// TIA Portal project "Project1" (V15.1)

(* hardware
DEVICE "S71500/ET200MP station_1"  S7-1500 station
   slot 0: "PS 25W 24VDC_1"  PS 25W 24VDC  6ES7 505-0KA00-0AB0  V1.0
   slot 0: "Rail_0"  Rack  6ES7 590-1***0-0AA0
   slot 1: "PLC_1"  CPU 1511-1 PN  6ES7 511-1AK00-0AB0  V1.8
      slot 3: "CPU display_1"  6ES7591-1AA00-0AA0
   slot 2: "DI 16x24VDC BA_1"  DI 16x24VDC BA  6ES7 521-1BH10-0AA0  V1.0
   slot 3: "DQ 8x230VAC/2A ST_1"  DQ 8x230VAC/2A ST  6ES7 522-5FF00-0AB0  V2.0
*)

// ===== PLC "PLC_1"  CPU 1511-1 PN =====

VAR_GLOBAL   // PLC tag table "Default tag table"
   "S1" AT %I0.0 : Bool;
   "S2" AT %I0.1 : Bool;
   "S3" AT %I0.2 : Bool;
   "L1" AT %Q0.0 : Bool;
END_VAR

ORGANIZATION_BLOCK "Main"   // OB1, FBD, ProgramCycle
TITLE = "Main Program Sweep (Cycle)"
{ S7_Optimized_Access := 'TRUE' }
VERSION : 0.1
   VAR_INPUT
      Initial_Call : Bool;   // Initial call of this OB
      Remanence : Bool;   // =True, if remanent data are available
   END_VAR
BEGIN

REGION Network 1
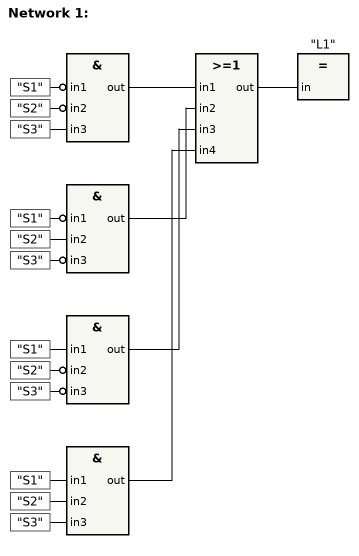
   "L1" := (NOT "S1" AND NOT "S2" AND "S3") OR (NOT "S1" AND "S2" AND NOT "S3") OR ("S1" AND NOT "S2" AND NOT "S3") OR ("S1" AND "S2" AND "S3");
END_REGION
END_ORGANIZATION_BLOCK